TYPE ST_Parameters :
STRUCT
	fCyclicTime 						: LREAL := 0.01; //[s]
	fMaxVelocityLimit 					: LREAL := 0.05; //[m/s]
	stOpenLoopControlSettings 			: ST_OpenLoopControlSettings;
	stClosedLoopControlSettings 		: ST_ClosedLoopControlSettings;
	stPressureFeedback 					: ST_ActiveDamping;
END_STRUCT
END_TYPE

(* stored: Version 1.1.0.1, ProductVersion 3.1.4024.10
   DUT ST_Parameters: Id {0acdc32a-38d7-42ed-a023-5b5f43624fa6} *)
